DATA_BLOCK "CalcVolume_Tank4_DB"
{ S7_Optimized_Access := 'FALSE' }
VERSION : 0.1
"CalculationVolume"

BEGIN
   IW_Radius := 1.468;
   IW_ValueFromSensor := 13.19083;
   IW_K_for_Tonnag := 1.35;
   IW_K_for_Level := 1.35;
   QW_Volume := 66.11805;
   QW_Tonnag := 89.25937;
   QW_RealLevel := 9.770983;
   sW_S := 6.766776;
   sW_Volume := 66.11805;
   sW_RealLevel := 9.770983;

END_DATA_BLOCK

